{attribute 'linkalways'} 
{attribute 'no_explicit_call' := 'This FB is a CLASS and must be accessed using methods or properties'}
{attribute 'enable_dynamic_creation'}
FUNCTION_BLOCK Node_ContainerType_Vector_TcVnVector3_UINT EXTENDS Node
VAR
    out : _GUID;
END_VAR

METHOD PUBLIC  Clone : I_Node
VAR
	pNode : POINTER TO Node_ContainerType_Vector_TcVnVector3_UINT;
END_VAR
pNode := __NEW(Node_ContainerType_Vector_TcVnVector3_UINT);
Clone := pNode^;
END_METHOD

METHOD FB_init : BOOL
VAR_INPUT
	bInitRetains : BOOL; // if TRUE, the retain variables are initialized (warm start / cold start)
	bInCopyCode : BOOL;  // if TRUE, the instance afterwards gets moved into the copy code (online change)
END_VAR
AddOutput('out', out);
END_METHOD

METHOD PROTECTED OnExecute
out.Value := ContainerType_Vector_TcVnVector3_UINT;
END_METHOD

END_FUNCTION_BLOCK

(* stored: Version 1.1.0.1, ProductVersion 3.1.4026.17
   POU Node_ContainerType_Vector_TcVnVector3_UINT: Id {b3b970de-5c8e-01f0-2c5c-77cb8960f826}, SpecialFunc None
   Folder Constructor: Id {a2e5e9fa-92f6-02e5-350d-bc4aab7f80f4}
   Method Clone: Id {2603a67c-0e8e-0f85-3411-9f0f2f8dd07f}
   Method FB_init: Id {c687cfdc-7f1e-04ce-1cd9-4f42d57cb4ea}
   Method OnExecute: Id {beeafc65-d1bd-094a-1ba8-10d62bf46984} *)
